Fanuc TP program (LS listing): testfold.ls

/PROG  TESTFOLD
/ATTR
OWNER		= MNEDITOR;
COMMENT		= "";
PROG_SIZE	= 295;
CREATE		= DATE 17-04-20  TIME 09:55:56;
MODIFIED	= DATE 17-04-20  TIME 10:31:54;
FILE_NAME	= ;
VERSION		= 0;
LINE_COUNT	= 2;
MEMORY_SIZE	= 675;
PROTECT		= READ_WRITE;
TCD:  STACK_SIZE	= 0,
      TASK_PRIORITY	= 50,
      TIME_SLICE	= 0,
      BUSY_LAMP_OFF	= 0,
      ABORT_REQUEST	= 0,
      PAUSE_REQUEST	= 0;
DEFAULT_GROUP	= *,*,*,*,*;
CONTROL_CODE	= 00000000 00000000;
/APPL
  ARC : TRUE ;
  ARC Welding Equipment : 1,*,*,*,*;

MPAS ;
MPAS_NUM_PASSES        : 0;
MPAS_LAST_PASS         : 0;
MPAS_CURRENT_PASS      : 0;
MPAS_STATUS_PASS       : 0;
/MN
   1:  CALL FOLD3    ;
   2:  CALL UNFOLD3    ;
/POS
/END
